{attribute 'qualified_only'}
VAR_GLOBAL
	start_record : BOOL := FALSE;
END_VAR

(* stored: Version 1.1.0.1, ProductVersion 3.1.4024.12
   GVL GVL_Visu: Id {d5c40656-8b70-45f0-857c-7eec9b3104e8} *)
